{attribute 'GeneratedUsingTerminal: EL1202-0100-0016'}
{attribute addProperty BoxType "EL1202-0100-0016"}
{attribute addProperty Id "Channel_1AT %I*Channel_830843C11Channel_2AT %I*Channel_830843C11ReservedEMPTY_STRUCTURE0DCAT %I*DC_1A6E66258WcStateAT %I*WcState_9091E0EB2InfoDataAT %I*InfoData_A7436BC610"}
{attribute addProperty CRC "1685997063"}
{attribute addProperty Size "22"}
TYPE EL1202_647E4607 EXTENDS EtcSlaveTerminalBase_947E5A46 :
STRUCT
	{attribute addProperty Name "Channel_1"}
	Channel_1 : Channel_830843C1;
	{attribute addProperty Name "Channel_2"}
	Channel_2 : Channel_830843C1;
	{attribute addProperty Name "Reserved"}
	Reserved : EMPTY_STRUCTURE;
	{attribute addProperty Name "DC"}
	DC : DC_1A6E6625;
	{attribute addProperty Name "WcState"}
	WcState : WcState_9091E0EB;
	{attribute addProperty Name "InfoData"}
	InfoData : InfoData_A7436BC6;
END_STRUCT
END_TYPE

(* stored: Version 1.2.0.0, ProductVersion 3.1.4024.9
   DUT EL1202_647E4607: Id {3591b0ad-800d-484d-a0ae-ddaccfd596c3} *)
